TYPE ST_CMD_EPICS :
STRUCT
	
	bExecute:BOOL:=FALSE;
	bEnable:BOOL:=FALSE;
	bReset:BOOL:=FALSE;
	fVelSet:LREAL:=0;
	fPosSet:LREAL:=0;
	eTargetStateCmd: TARGET_STATE_MACHINE:=0;
	
	//brake
	bBrakeLockOnCmd:BOOL:=FALSE;
	bFreeWheelOnOnCmd:BOOL:=TRUE;
	fBrakeSpNm:LREAL:=0;
END_STRUCT
END_TYPE

(* stored: Version 1.1.0.1, ProductVersion 3.1.4022.6
   DUT ST_CMD_EPICS: Id {4efa13fc-0f5c-44cc-8a6d-b3a9305f00ac} *)
